(* IEC 61131-3 sources: Laboratorijsko-busace-postrojenje/Libraries/DRV_mbus, 2 files *)

(* ---- DRV_mbus.fun ---- *)
(********************************************************************
 * COPYRIGHT (C) BERNECKER + RAINER, AUSTRIA, A-5142 EGGELSBERG
 ********************************************************************
 * Library: DRV_mbus
 * File: DRV_mbus.fun
 * Created: 11.11.2003
 ********************************************************************
 * Functions and function blocks of library DRV_mbus
 ********************************************************************)
FUNCTION_BLOCK MBMCmd				(*operates the modbus protocol in runtime*)
	VAR_INPUT
		enable	:BOOL;				(*enables execution*)
		ident	:UDINT;				(*identifier of the MBMOpen() FBK*)
		mfc	:USINT;					(*modbus function call*)
		node	:USINT;				(*station number (0 = broadcast)*)
		data	:UDINT;				(*pointer to the data area*)
		offset	:UINT;				(*offset*)
		len	:UINT;					(*size of data*)
	END_VAR
	VAR_OUTPUT
		status	:UINT;				(*execution status: ERR_OK, ERR_FUB_ENABLE_FALSE, 0xXXXX = see help*)
	END_VAR
END_FUNCTION_BLOCK

FUNCTION_BLOCK MBMClose				(*closes the driver environment to enable the MBMOpen() FBK to be called again*)
	VAR_INPUT
		enable	:BOOL;				(*enables execution*)
		ident	:UDINT;				(*identifier of the MBMOpen() FBK*)
	END_VAR
	VAR_OUTPUT
		status	:UINT;				(*execution status: ERR_OK, ERR_FUB_ENABLE_FALSE, 0xXXXX = see help*)
	END_VAR
END_FUNCTION_BLOCK

FUNCTION_BLOCK MBMaster				(*operates the modbus protocol in runtime*)
	VAR_INPUT
		enable	:BOOL;				(*enables execution*)
		ident	:UDINT;				(*identifier of the MBMOpen() FBK*)
	END_VAR
	VAR_OUTPUT
		status	:UINT;				(*execution status: ERR_OK, ERR_FUB_ENABLE_FALSE, 0xXXXX = see help*)
		execute	:BOOL;				(*command executed (execute = 1)*)
		recordnum	:UINT;			(*number of the entry in the data object currently being processed*)
	END_VAR
END_FUNCTION_BLOCK

FUNCTION_BLOCK MBMOpen				(*configures the interface and initializes the internal structures that are required*)
	VAR_INPUT
		enable	:BOOL;				(*enables execution*)
		pDevice	:UDINT;				(*device name given as a pointer*)
		pMode	:UDINT;				(*pointer to the mode description string*)
		pConfig	:UDINT;				(*pointer to the data object name*)
		timeout	:UINT;				(*response timeout in milliseconds (the value must be a multiple of 10)*)
		ascii	:USINT;				(*modBus mode (0 = RTU / 1 = ASCII)*)
	END_VAR
	VAR_OUTPUT
		status	:UINT;				(*execution status: ERR_OK, ERR_FUB_ENABLE_FALSE, 0xXXXX = see help*)
		ident	:UDINT;				(*identifier for the MBMaster(), MBMCmd() and MBMClose() FBKs*)
	END_VAR
END_FUNCTION_BLOCK

FUNCTION_BLOCK MBSClose				(*closes the driver environment to enable the MBSOpen() FBK to be called again*)
	VAR_INPUT
		enable	:BOOL;				(*enables execution*)
		ident	:UDINT;				(*identifier of the MBSOpen() FBK*)
	END_VAR
	VAR_OUTPUT
		status	:UINT;				(*execution status: ERR_OK, ERR_FUB_ENABLE_FALSE, 0xXXXX = see help*)
	END_VAR
	VAR
		InitCount	:USINT;			(*internal variable*)
	END_VAR
END_FUNCTION_BLOCK

FUNCTION_BLOCK MBSlave				(*operates the modbus protocol in runtime*)
	VAR_INPUT
		enable	:BOOL;				(*enables execution*)
		ident	:UDINT;				(*identifier of the MBSOpen() FBK*)
	END_VAR
	VAR_OUTPUT
		status	:UINT;				(*execution status: ERR_OK, ERR_FUB_ENABLE_FALSE, 0xXXXX = see help*)
		exec	:UINT;				(*counter for modbus commands received*)
	END_VAR
END_FUNCTION_BLOCK

FUNCTION_BLOCK MBSOpen				(*configures the interface and initializes the internal structures that are required*)
	VAR_INPUT
		enable	:BOOL;				(*enables execution*)
		pDevice	:UDINT;				(*device name given as a pointer*)
		pMode	:UDINT;				(*pointer to the mode description string*)
		pCoilStat	:UDINT;			(*pointer to the coil status (modbus simulation variable)*)
		pInputStat	:UDINT;			(*pointer to the input status (modbus simulation variable)*)
		pHoldingReg	:UDINT;			(*pointer to the holding register (modbus simulation variable)*)
		pInputReg	:UDINT;			(*pointer to the input register (modbus simulation variable)*)
		own_ID	:USINT;				(*own node number*)
		timeout	:UINT;				(*response timeout in milliseconds (the value must be a multiple of 10)*)
	END_VAR
	VAR_OUTPUT
		status	:UINT;				(*execution status: ERR_OK, ERR_FUB_ENABLE_FALSE, 0xXXXX = see help*)
		ident	:UDINT;				(*identifier for the MBClient() and MBSClose() FBKs*)
	END_VAR
	VAR
		FirstInit	:UDINT;			(*internal variable*)
		InitCount	:USINT;			(*internal variable*)
	END_VAR
END_FUNCTION_BLOCK

(* ---- DRV_mbus.var ---- *)
(********************************************************************
 * COPYRIGHT (C) BERNECKER + RAINER, AUSTRIA, A-5142 EGGELSBERG
 ********************************************************************
 * Library: DRV_mbus
 * File: DRV_mbus.var
 * Created: 11.11.2003
 ********************************************************************
 * Constants of library DRV_mbus
 ********************************************************************)
VAR CONSTANT
	mbERR_INVALID_PARAM	: UINT	:= 20201;	(*invalid FBK parameter (e.g. pDevice = 0)*)
	mbERR_ILG_O_NODE_N	: UINT	:= 20205;	(*invalid own_ID stated in MBSOpen() FBK; valid IDs are between 1 and 247*)
	mbERR_ILG_IDENT	: UINT	:= 20210;		(*invalid ID or ID is 0*)
	mbERR_ILG_MBVAR	: UINT	:= 20215;		(*ModBus simulation variable invalid or missing (MBSOpen() and MBSlave() FBK)*)
	mbERR_NODE_TOUT	: UINT	:= 20220;		(*in MBSOpen(), MBMOpen(): invalid value for timeout parameter, in MBMCmd(), MBMaster(), MBSlave(): timeout detected*)
	mbERR_CMD_ENTRY	: UINT	:= 20240;		(*invalid entry in data object, invalid length of data object*)
	mbERR_CMD_NULL	: UINT	:= 20241;		(*data object not present or data parameter in MBMCmd FBK is 0*)
	mbERR_CMD_EVENTPV	: UINT	:= 20242;	(*invalid EventPV stated in the data object*)
	mbERR_CMD_FUNCTION	: UINT	:= 20243;	(*invalid ModBus function stated in the data object or in the MBMCmd() FBK*)
	mbERR_CMD_NODE	: UINT	:= 20244;		(*invalid nodenumber stated in the data object or in the MBMCmd() FBK*)
	mbERR_CMD_LOCALPV	: UINT	:= 20245;	(*invalid EventPV stated in the data object*)
	mbERR_CMD_LENGTH	: UINT	:= 20246;	(*invalid length stated in the data object*)
	mbERR_NO_MEM	: UINT	:= 20250;		(*no memory for internal library management*)
	mbERR_MEM_FREE	: UINT	:= 20252;		(*memory for internal library management cannot be freed*)
	mbERR_RESP_ERROR	: UINT	:= 20260;	(*invalid frame received*)
	mbERR_RESP_LENGTH	: UINT	:= 20261;	(*frame with wrong length received*)
	mbERR_RESP_INVALID	: UINT	:= 20262;	(*error in frame*)
	mbERR_RESP_CRC	: UINT	:= 20263;		(*error in frame check (CRC / LRC) MBMaster() and MBMCmd()*)
	mbERR_QUERY_CRC	: UINT	:= 20264;		(*error in frame check (CRC) MBMSlave()*)
	mbERR_FRM_READ	: UINT	:= 20291;		(*error while receiving a frame (FRM_read())*)
	mbERR_FRM_GETBUF	: UINT	:= 20292;	(*no write buffer available (FRM_gbuf())*)
	mbERR_FRM_WRITE	: UINT	:= 20293;		(*error while writing a frame (FRM_write())*)
	mbERR_FRM_RELOUTBUF	: UINT	:= 20294;	(*error in buffer return (FRM_robuf())*)
	mbERR_FRM_RELBUF	: UINT	:= 20295;	(*error in buffer return (FRM_rbuf())*)
	mbERR_FRM_CLOSE	: UINT	:= 20296;		(*error while closing the interface (FRM_close())*)
END_VAR
